(* IEC 61131-3 sources: Elmo_Master/Lasal_PRG/Elmo_EtherCAT_Test_4Axis/Class/LMCDiagnosticsService (part 3) *)

			32:
				mailboxResult := InputLatch.SubmitDs402HomeControl(
					OperationToken:=Ds402HomeState[101]$UDINT,
					AxisReference:=axisReference, Command:=4);
				if mailboxResult = 0 then
					Ds402HomeState[117] := 0;
					Ds402HomeState[112] := currentCycle$DINT;
					Ds402HomeState[92] := 34;
				elsif mailboxResult = 1 then
					Ds402HomeState[92] := 33;
				else
					failure := TRUE;
					failureDetail := 11;
					failureNative := TO_UDINT(0 - mailboxResult);
				end_if;

			33:
				mailboxResult := InputLatch.GetDs402HomeControlState(
					OperationToken:=Ds402HomeState[101]$UDINT);
				if mailboxResult = 0 then
					Ds402HomeState[117] := 0;
					Ds402HomeState[112] := currentCycle$DINT;
					Ds402HomeState[92] := 34;
				elsif mailboxResult <> 1 then
					failure := TRUE;
					failureDetail := 11;
					failureNative := TO_UDINT(0 - mailboxResult);
				end_if;

			34:
				if newCycle &
					(currentCycle <> Ds402HomeState[112]$UDINT) then
					if (Ds402HomeState[94] <> 0) |
						(Ds402HomeState[113] <> 0) |
						(Ds402HomeState[116] <> 0) |
						(Ds402HomeState[117] <> 0) |
						(Ds402HomeState[127] <> 0) |
						((statusWord and 0x0008) <> 0) |
						((statusWord and 0x2000) <> 0) |
						((baseState <> 0x0040) & (baseState <> 0x0021) &
						 (baseState <> 0x0023) & (baseState <> 0x0027)) |
						(actualPosition <> 0) then
						failure := TRUE;
						failureNative := 24;
					else
						Ds402HomeState[106] := 2;
						Ds402HomeState[107] := 0;
						Ds402HomeState[108] := 0;
						Ds402HomeState[recordBase + 14] := 0;
						Ds402HomeState[recordBase + 15] := 0;
						Ds402HomeState[recordBase + 16] := 0;
						Ds402HomeState[recordBase + 20] := currentCycle$DINT;
						Ds402HomeState[recordBase + 21] := 0;
						ownerResult := -1;
						if IsClientConnected(#AxisOwnership) then
							ownerResult :=
								AxisOwnership.PublishAxisOwnershipDs402Receipt(
								AxisMask:=axisMask,
								AdmissionToken:=admissionToken,
								OwnerGeneration:=ownerGeneration,
								ReportKind:=
									LMC_DIAG_OWNER_REPORT_TERMINAL_SUCCESS,
								ReportValue0:=0,
								ReportValue1:=0,
								ObservationCycle:=currentCycle,
								pDs402State:=#Ds402HomeState[0],
								Ds402StateSize:=sizeof(Ds402HomeState));
						end_if;
						if ownerResult = 0 then
							Ds402HomeState[125] := 2;
							ownerResult :=
								AxisOwnership.PublishAxisOwnershipDs402Receipt(
									AxisMask:=axisMask,
									AdmissionToken:=admissionToken,
									OwnerGeneration:=ownerGeneration,
									ReportKind:=
										LMC_DIAG_OWNER_REPORT_TERMINAL_SUCCESS,
									ReportValue0:=0,
									ReportValue1:=0,
									ObservationCycle:=currentCycle,
									pDs402State:=#Ds402HomeState[0],
									Ds402StateSize:=sizeof(Ds402HomeState));
							if ownerResult = 1 then
								Ds402HomeState[92] :=
									LMC_DIAG_DS402_STAGE_FINALIZE;
							elsif ownerResult <> 0 then
								Ds402HomeState[92] := 101;
							end_if;
							RETURN;
						elsif ownerResult = 1 then
							Ds402HomeState[92] := LMC_DIAG_DS402_STAGE_FINALIZE;
							RETURN;
						else
							Ds402HomeState[92] := 101;
						end_if;
					end_if;
				end_if;
		end_case;
	end_if;

	// SDO start stages use one persistent executor at a time.
	stage := Ds402HomeState[92];
	startSdo := FALSE;
	sdoIsWrite := FALSE;
	sdoIndex := 0;
	homeSdoSubIndex := 0;
	sdoLength := 0;
	sdoData := 0;
	nextStage := stage;
	if (failure = FALSE) & (stage < 90) then
		case stage of
			2:
				startSdo := TRUE; sdoIndex := 0x6061;
				sdoLength := 1; nextStage := 3;
			4:
				startSdo := TRUE; sdoIsWrite := TRUE; sdoIndex := 0x607C;
				sdoLength := 4; sdoData := Ds402HomeState[recordBase + 10]$UDINT;
				nextStage := 5;
			6:
				startSdo := TRUE; sdoIsWrite := TRUE; sdoIndex := 0x6098;
				sdoLength := 1; sdoData := Ds402HomeState[recordBase + 9]$UDINT;
				nextStage := 7;
			16:
				startSdo := TRUE; sdoIsWrite := TRUE; sdoIndex := 0x6060;
				sdoLength := 1; sdoData := 6; nextStage := 17;
			18:
				startSdo := TRUE; sdoIndex := 0x6061;
				sdoLength := 1; nextStage := 19;
			28:
				startSdo := TRUE; sdoIsWrite := TRUE; sdoIndex := 0x6060;
				sdoLength := 1; sdoData := 8; nextStage := 29;
			30:
				startSdo := TRUE; sdoIndex := 0x6061;
				sdoLength := 1; nextStage := 31;
		end_case;
	end_if;

	if startSdo then
		if IsClientConnected(#AxisOwnership) = FALSE then
			failure := TRUE;
			failureNative := 24;
		else
			ownerResult := AxisOwnership.ValidateAxisOwnership(
				CommandId:=0x7D15,
				Reference:=axisReference,
				ExpectedAxisMask:=axisMask,
				OwnerKind:=LMC_DIAG_OWNER_KIND_DS402_HOME,
				ResourceKind:=LMC_DIAG_RESOURCE_DS402_HOME,
				AdmissionMode:=LMC_DIAG_ADMISSION_LIFECYCLE,
				CallerSessionEpoch:=ds402ProcessOwnerSessionEpoch,
				RequestSequence:=ownerRequestSequence,
				AdmissionToken:=admissionToken,
				OwnerGeneration:=ownerGeneration,
				RequiredPhase:=LMC_DIAG_OWNER_PHASE_ACTIVE);
			if ownerResult <> 0 then
				failure := TRUE;
				failureNative := TO_UDINT(0 - ownerResult);
			elsif Ds402HomeState[126] = 0 then
					ownerResult := AxisOwnership.PublishAxisOwnership(
						AxisMask:=axisMask,
						AdmissionToken:=admissionToken,
						OwnerGeneration:=ownerGeneration,
						ReportKind:=LMC_DIAG_OWNER_REPORT_DISPATCH,
						ReportValue0:=TO_UDINT(sdoIndex),
						ReportValue1:=Ds402HomeState[101]$UDINT,
						ObservationCycle:=currentCycle);
				if ownerResult = 0 then
					Ds402HomeState[126] := 1;
				else
					failure := TRUE;
					failureNative := TO_UDINT(0 - ownerResult);
				end_if;
			end_if;
		end_if;
	end_if;

	if startSdo & (failure = FALSE) then
		executorConnected := FALSE;
		executorReusable := FALSE;
		case axisReference of
			1:
				executorConnected := IsClientConnected(#SdoAxis1) <> 0;
				if executorConnected then
					executorReusable := SdoAxis1.IsReusable();
				end_if;
			2:
				executorConnected := IsClientConnected(#SdoAxis2) <> 0;
				if executorConnected then
					executorReusable := SdoAxis2.IsReusable();
				end_if;
			3:
				executorConnected := IsClientConnected(#SdoAxis3) <> 0;
				if executorConnected then
					executorReusable := SdoAxis3.IsReusable();
				end_if;
			4:
				executorConnected := IsClientConnected(#SdoAxis4) <> 0;
				if executorConnected then
					executorReusable := SdoAxis4.IsReusable();
				end_if;
		end_case;
		if (executorConnected = FALSE) | (executorReusable = FALSE) then
			failure := TRUE;
			failureNative := 24;
		else
			sdoToken := Ds402HomeState[99]$UDINT + 1;
			if sdoToken = 0 then
				sdoToken := 1;
			end_if;
			Ds402HomeState[99] := sdoToken$DINT;
			Ds402HomeState[95] := 0;
			if sdoIsWrite then
				Ds402HomeState[95] := 1;
			end_if;
			Ds402HomeState[96] := sdoIndex$DINT;
			Ds402HomeState[97] := homeSdoSubIndex$DINT;
			Ds402HomeState[98] := sdoLength$DINT;
			Ds402HomeState[100] := sdoData$DINT;
			startCycle := Ds402HomeState[recordBase + 19]$UDINT;
			timeoutMs := Ds402HomeState[recordBase + 13]$UDINT;
			elapsedCycles := serviceNow - serviceStart;
			remainingMs := 1;
			if elapsedCycles < timeoutMs then
				remainingMs := timeoutMs - elapsedCycles;
			end_if;
			if remainingMs > 60000 then
				remainingMs := 60000;
			end_if;
			startResult := ERROR;
			case axisReference of
				1:
					if sdoIsWrite then
						startResult := SdoAxis1.TryStartWrite(sdoToken, sdoIndex,
							homeSdoSubIndex, (#sdoData)$^USINT, sdoLength, remainingMs);
					else
						startResult := SdoAxis1.TryStartRead(sdoToken, sdoIndex,
							homeSdoSubIndex, sdoLength, remainingMs);
					end_if;
				2:
					if sdoIsWrite then
						startResult := SdoAxis2.TryStartWrite(sdoToken, sdoIndex,
							homeSdoSubIndex, (#sdoData)$^USINT, sdoLength, remainingMs);
					else
						startResult := SdoAxis2.TryStartRead(sdoToken, sdoIndex,
							homeSdoSubIndex, sdoLength, remainingMs);
					end_if;
				3:
					if sdoIsWrite then
						startResult := SdoAxis3.TryStartWrite(sdoToken, sdoIndex,
							homeSdoSubIndex, (#sdoData)$^USINT, sdoLength, remainingMs);
					else
						startResult := SdoAxis3.TryStartRead(sdoToken, sdoIndex,
							homeSdoSubIndex, sdoLength, remainingMs);
					end_if;
				4:
					if sdoIsWrite then
						startResult := SdoAxis4.TryStartWrite(sdoToken, sdoIndex,
							homeSdoSubIndex, (#sdoData)$^USINT, sdoLength, remainingMs);
					else
						startResult := SdoAxis4.TryStartRead(sdoToken, sdoIndex,
							homeSdoSubIndex, sdoLength, remainingMs);
					end_if;
			end_case;
			if startResult = READY then
				// Once the mode-6 write is accepted, cleanup must assume it may
				// have reached the drive even if its callback is later lost.
				if stage = 16 then
					Ds402HomeState[116] := 1;
				end_if;
				Ds402HomeState[94] := 1;
				Ds402HomeState[92] := nextStage;
			else
				failure := TRUE;
				failureNative := 24;
			end_if;
		end_if;
	end_if;

	stage := Ds402HomeState[92];
	waitSdo := (stage = 3) | (stage = 5) | (stage = 7) |
		(stage = 17) | (stage = 19) | (stage = 29) | (stage = 31);
	if (failure = FALSE) & waitSdo then
		completionResult := -2;
		case axisReference of
			1:
				if IsClientConnected(#SdoAxis1) then
					completionResult := SdoAxis1.CopyCompletion(
						Ds402HomeState[99]$UDINT, #completion, sizeof(completion));
				end_if;
			2:
				if IsClientConnected(#SdoAxis2) then
					completionResult := SdoAxis2.CopyCompletion(
						Ds402HomeState[99]$UDINT, #completion, sizeof(completion));
				end_if;
			3:
				if IsClientConnected(#SdoAxis3) then
					completionResult := SdoAxis3.CopyCompletion(
						Ds402HomeState[99]$UDINT, #completion, sizeof(completion));
				end_if;
			4:
				if IsClientConnected(#SdoAxis4) then
					completionResult := SdoAxis4.CopyCompletion(
						Ds402HomeState[99]$UDINT, #completion, sizeof(completion));
				end_if;
		end_case;
		if completionResult = 0 then
			Ds402HomeState[94] := 0;
			if (completion.ValidationCode <> 0) | (completion.OsResult <> 0) |
				(completion.AbortCode <> 0) |
				(completion.ObjectIndex <> Ds402HomeState[96]$UINT) |
				(completion.SubIndex <> Ds402HomeState[97]$USINT) |
				(completion.ActualLength <> Ds402HomeState[98]$UDINT) |
				(completion.IsWrite <> Ds402HomeState[95]$USINT) then
				failure := TRUE;
				if completion.AbortCode <> 0 then
					failureNative := completion.AbortCode;
				elsif completion.OsResult <> 0 then
					failureNative := completion.OsResult$UDINT;
				else
					failureNative := completion.ValidationCode;
				end_if;
			else
				case stage of
					3:
						if (completion.Data and 0xFF) <> 8 then
							failure := TRUE; failureNative := completion.Data;
						else
							Ds402HomeState[105] := 8; Ds402HomeState[92] := 4;
						end_if;
					5: Ds402HomeState[92] := 6;
					7: Ds402HomeState[92] := 14;
					17:
						Ds402HomeState[116] := 1; Ds402HomeState[92] := 18;
					19:
						if (completion.Data and 0xFF) <> 6 then
							failure := TRUE; failureNative := completion.Data;
						else
							Ds402HomeState[92] := 20;
						end_if;
					29: Ds402HomeState[92] := 30;
					31:
						if (completion.Data and 0xFF) <> 8 then
							failure := TRUE; failureNative := completion.Data;
						else
							Ds402HomeState[116] := 0; Ds402HomeState[92] := 32;
						end_if;
				end_case;
			end_if;
		elsif (completionResult <> -2) & (completionResult <> -3) then
			failure := TRUE;
			failureNative := TO_UDINT(0 - completionResult);
		end_if;
	end_if;

	if failure then
		if Ds402HomeState[94] <> 0 then
			orphanResult := -1;
			case axisReference of
				1:
					if IsClientConnected(#SdoAxis1) then
						orphanResult := SdoAxis1.MarkOrphan(Ds402HomeState[99]$UDINT);
					end_if;
				2:
					if IsClientConnected(#SdoAxis2) then
						orphanResult := SdoAxis2.MarkOrphan(Ds402HomeState[99]$UDINT);
					end_if;
				3:
					if IsClientConnected(#SdoAxis3) then
						orphanResult := SdoAxis3.MarkOrphan(Ds402HomeState[99]$UDINT);
					end_if;
				4:
					if IsClientConnected(#SdoAxis4) then
						orphanResult := SdoAxis4.MarkOrphan(Ds402HomeState[99]$UDINT);
					end_if;
			end_case;
			// -2 can mean that the exact result won the timeout race. Keep the
			// executor in the cleanup drain path so a ready result is consumed.
			if (orphanResult = 0) | (orphanResult = -2) then
				Ds402HomeState[94] := 0;
				Ds402HomeState[113] := 1;
				Ds402HomeState[127] := 0;
			else
				// Keep the pending token and remember that exact retirement failed.
				Ds402HomeState[127] := 1;
			end_if;
		end_if;
		if preemptionCleanup then
			Ds402HomeState[106] := 4;
		else
			Ds402HomeState[106] := 3;
		end_if;
		Ds402HomeState[107] := failureDetail$DINT;
		Ds402HomeState[108] := failureNative$DINT;
		Ds402HomeState[112] := currentCycle$DINT;
		Ds402HomeState[119]$UDINT := serviceNow;
		Ds402HomeState[92] := 90;
		RETURN;
	end_if;

	// Failure cleanup attempts bit 4 low, setpoint alignment, CSP restore and RT
	// release. Timeout never claims that any of those cleanup steps completed.
	stage := Ds402HomeState[92];
	if stage < 90 then
		RETURN;
	end_if;
	if preemptionCleanup then
		HandleAxisDs402HomeCleanupStages(
			Stage:=stage,
			AxisReference:=axisReference,
			AxisMask:=axisMask,
			AdmissionToken:=admissionToken,
			OwnerGeneration:=ownerGeneration,
			Ds402ProcessOwnerSessionEpoch:=ds402ProcessOwnerSessionEpoch,
			OwnerRequestSequence:=ownerRequestSequence,
			SafetyAdmissionToken:=safetyAdmissionToken,
			SafetyOwnerGeneration:=safetyOwnerGeneration,
			InitialCurrentCycle:=currentCycle,
			ServiceNow:=serviceNow,
			ActualPosition:=actualPosition,
			PreemptionCleanup:=TRUE);
	else
		HandleAxisDs402HomeCleanupStages(
			Stage:=stage,
			AxisReference:=axisReference,
			AxisMask:=axisMask,
			AdmissionToken:=admissionToken,
			OwnerGeneration:=ownerGeneration,
			Ds402ProcessOwnerSessionEpoch:=ds402ProcessOwnerSessionEpoch,
			OwnerRequestSequence:=ownerRequestSequence,
			SafetyAdmissionToken:=0,
			SafetyOwnerGeneration:=0,
			InitialCurrentCycle:=currentCycle,
			ServiceNow:=serviceNow,
			ActualPosition:=actualPosition,
			PreemptionCleanup:=FALSE);
	end_if;

END_FUNCTION

FUNCTION LMCDiagnosticsService::HandleAxisDs402HomeReceiptStages
	VAR_INPUT
		Stage 	: DINT;
	END_VAR
	VAR_OUTPUT
		Result 	: DINT;
	END_VAR
	VAR
		activeIndex, recordBase : DINT;
		axisReference : UINT;
		axisMask, admissionToken, ownerGeneration : UDINT;
		ds402ProcessOwnerSessionEpoch, ownerRequestSequence : UDINT;
		receiptGeneration : UDINT;
		ownerResult, receiptResult, receiptKind, receiptPhase : DINT;
		terminalRecordState : DINT;
	END_VAR

	Result := 1;
	if stage = LMC_DIAG_DS402_STAGE_INTENT_DISCARD_CLEAR then
		activeIndex := Ds402HomeState[93];
		if (activeIndex < 0) | (activeIndex > 3) |
			(sizeof(Ds402HomeState) <> 512) then
			Ds402HomeState[92] := 101;
			RETURN;
		end_if;
		recordBase := activeIndex * 23;
		// Stage 86 keeps the axis selector authoritative until this idempotent
		// record clear is complete. Runtime WAL bytes remain invalid under stage 0
		// and are replaced by the next preflight.
		_memset(dest:=#Ds402HomeState[recordBase], usByte:=0, cntr:=92);
		Ds402HomeState[92] := 0;
		RETURN;
	end_if;
	if stage = LMC_DIAG_DS402_STAGE_RESERVE_INTENT then
		activeIndex := Ds402HomeState[93];
		if (activeIndex < 0) | (activeIndex > 3) |
			(sizeof(Ds402HomeState) <> 512) then
			Ds402HomeState[92] := 101;
			RETURN;
		end_if;
		recordBase := activeIndex * 23;
		axisMask := TO_UDINT(1) shl TO_UDINT(activeIndex);
		if IsClientConnected(#AxisOwnership) = FALSE then
			RETURN;
		end_if;
		// Tokenless mode is confined to stage 87 rollback resolution. The
		// provider either adopts one exact RESERVED tuple, proves absence/later
		// ownership, or leaves the intent fail-closed.
		receiptResult := AxisOwnership.PublishAxisOwnershipDs402Receipt(
			AxisMask:=axisMask,
			AdmissionToken:=0,
			OwnerGeneration:=0,
			ReportKind:=LMC_DIAG_DS402_RECEIPT_ROLLBACK,
			ReportValue0:=0,
			ReportValue1:=0,
			ObservationCycle:=Ds402HomeState[118]$UDINT,
			pDs402State:=#Ds402HomeState[0],
			Ds402StateSize:=sizeof(Ds402HomeState));
		if receiptResult = 1 then
			// Commit record cleanup before touching any selector or WAL byte.
			Ds402HomeState[92] :=
				LMC_DIAG_DS402_STAGE_INTENT_DISCARD_CLEAR;
		elsif receiptResult = 2 then
			// Preserve only an untouched raw tombstone. Once adoption or the record
			// bridge was published, commit a durable record-clear cleanup first.
			if (Ds402HomeState[119]$UDINT =
				LMC_DIAG_DS402_INTENT_ADOPT_MAGIC) |
				(Ds402HomeState[recordBase] = 1) then
				Ds402HomeState[92] :=
					LMC_DIAG_DS402_STAGE_INTENT_DISCARD_CLEAR;
			elsif Ds402HomeState[recordBase]$UDINT <>
				Ds402HomeState[115]$UDINT then
				Ds402HomeState[92] := 101;
				RETURN;
			else
				// No local record changed. Stage 0 invalidates the retained WAL in one
				// commit; the next preflight overwrites it before reuse.
				Ds402HomeState[92] := 0;
			end_if;
		elsif receiptResult = -1 then
			// A transient result retains the durable intent indefinitely.
		elsif receiptResult <> 0 then
			Ds402HomeState[92] := 101;
		end_if;
		RETURN;
	end_if;
	if stage = 0 then
		RETURN;
	end_if;
	activeIndex := Ds402HomeState[93];
	admissionToken := Ds402HomeState[122]$UDINT;
	ownerGeneration := Ds402HomeState[123]$UDINT;
	if (activeIndex < 0) | (activeIndex > 3) |
		(sizeof(Ds402HomeState) <> 512) then
		Ds402HomeState[92] := 101;
		RETURN;
	end_if;
	recordBase := activeIndex * 23;
	axisMask := TO_UDINT(1) shl TO_UDINT(activeIndex);
	receiptPhase := Ds402HomeState[125];
	receiptGeneration := Ds402HomeState[127]$UDINT;

	if stage = LMC_DIAG_DS402_STAGE_FINALIZE then
		receiptKind := Ds402HomeState[126];
		if (Ds402HomeState[124]$UDINT <> LMC_DIAG_DS402_RECEIPT_MAGIC) |
			(receiptPhase <> LMC_DIAG_DS402_RECEIPT_COMPLETE) |
			(receiptGeneration = 0) |
			(receiptGeneration <> Ds402HomeState[109]$UDINT) |
			(admissionToken = 0) | (ownerGeneration = 0) then
			Ds402HomeState[92] := 101;
			RETURN;
		end_if;
		case receiptKind of
			LMC_DIAG_DS402_RECEIPT_ROLLBACK:
				if (Ds402HomeState[106] <> 0) |
					((Ds402HomeState[recordBase] <> 0) &
					 (Ds402HomeState[recordBase] <> 1)) |
					((Ds402HomeState[recordBase + 22]$UDINT <> 0) &
					 (Ds402HomeState[recordBase + 22]$UDINT <>
					  receiptGeneration)) then
					Ds402HomeState[92] := 101;
					RETURN;
				end_if;
				_memset(dest:=#Ds402HomeState[recordBase],
					usByte:=0, cntr:=92);
			LMC_DIAG_OWNER_REPORT_TERMINAL_SUCCESS,
			LMC_DIAG_OWNER_REPORT_TERMINAL_SAFE_FAILURE:
				terminalRecordState := Ds402HomeState[106];
				if (((receiptKind = LMC_DIAG_OWNER_REPORT_TERMINAL_SUCCESS) &
					  (terminalRecordState <> 2)) |
					 ((receiptKind =
					   LMC_DIAG_OWNER_REPORT_TERMINAL_SAFE_FAILURE) &
					  (terminalRecordState <> 3))) |
					(Ds402HomeState[recordBase + 22]$UDINT <>
					 receiptGeneration) |
					((Ds402HomeState[recordBase] <> 1) &
					 (Ds402HomeState[recordBase] <> terminalRecordState)) then
					Ds402HomeState[92] := 101;
					RETURN;
				end_if;
				Ds402HomeState[101] := 0;
				Ds402HomeState[recordBase] := terminalRecordState;
		else
			Ds402HomeState[92] := 101;
			RETURN;
		end_case;
		// The local lifecycle stage is the final publication word.
		Ds402HomeState[92] := 0;
		RETURN;
	end_if;

	if Ds402HomeState[124]$UDINT = LMC_DIAG_DS402_RECEIPT_MAGIC then
		if receiptGeneration = 0 then
			case stage of
				LMC_DIAG_DS402_STAGE_ROLLBACK_PREPARED:
					receiptKind := LMC_DIAG_DS402_RECEIPT_ROLLBACK;
				89: receiptKind := LMC_DIAG_DS402_RECEIPT_ROLLBACK;
				34: receiptKind := LMC_DIAG_OWNER_REPORT_TERMINAL_SUCCESS;
				100: receiptKind :=
					LMC_DIAG_OWNER_REPORT_TERMINAL_SAFE_FAILURE;
			else
				Ds402HomeState[92] := 101;
				RETURN;
			end_case;
		else
			receiptKind := Ds402HomeState[126];
		end_if;
		receiptResult := -1;
		if IsClientConnected(#AxisOwnership) = FALSE then
			RETURN;
		end_if;
		receiptResult := AxisOwnership.PublishAxisOwnershipDs402Receipt(
			AxisMask:=axisMask,
			AdmissionToken:=admissionToken,
			OwnerGeneration:=ownerGeneration,
			ReportKind:=TO_UINT(receiptKind),
			ReportValue0:=Ds402HomeState[107]$UDINT,
			ReportValue1:=Ds402HomeState[108]$UDINT,
			ObservationCycle:=Ds402HomeState[110]$UDINT,
			pDs402State:=#Ds402HomeState[0],
			Ds402StateSize:=sizeof(Ds402HomeState));
		if receiptResult = 0 then
			if Ds402HomeState[125] = LMC_DIAG_DS402_RECEIPT_PREPARED then
				Ds402HomeState[125] := 2;
			end_if;
			if IsClientConnected(#AxisOwnership) = FALSE then
				RETURN;
			end_if;
			receiptResult :=
				AxisOwnership.PublishAxisOwnershipDs402Receipt(
					AxisMask:=axisMask,
					AdmissionToken:=admissionToken,
					OwnerGeneration:=ownerGeneration,
					ReportKind:=TO_UINT(receiptKind),
					ReportValue0:=Ds402HomeState[107]$UDINT,
					ReportValue1:=Ds402HomeState[108]$UDINT,
					ObservationCycle:=Ds402HomeState[110]$UDINT,
					pDs402State:=#Ds402HomeState[0],
					Ds402StateSize:=sizeof(Ds402HomeState));
			if receiptResult = 1 then
				Ds402HomeState[92] := LMC_DIAG_DS402_STAGE_FINALIZE;
			elsif (receiptResult <> 0) & (receiptResult <> -1) then
				Ds402HomeState[92] := 101;
			end_if;
		elsif receiptResult = 1 then
			Ds402HomeState[92] := LMC_DIAG_DS402_STAGE_FINALIZE;
		elsif receiptResult <> -1 then
			Ds402HomeState[92] := 101;
		end_if;
		RETURN;
	end_if;

	if stage = LMC_DIAG_DS402_STAGE_ROLLBACK_PREPARED then
		// This state is rollback-only. It must never warm-resume into Commit.
		receiptResult := -1;
		if IsClientConnected(#AxisOwnership) = FALSE then
			RETURN;
		end_if;
		receiptResult := AxisOwnership.PublishAxisOwnershipDs402Receipt(
			AxisMask:=axisMask,
			AdmissionToken:=admissionToken,
			OwnerGeneration:=ownerGeneration,
			ReportKind:=LMC_DIAG_DS402_RECEIPT_ROLLBACK,
			ReportValue0:=0,
			ReportValue1:=0,
			ObservationCycle:=Ds402HomeState[110]$UDINT,
			pDs402State:=#Ds402HomeState[0],
			Ds402StateSize:=sizeof(Ds402HomeState));
		if receiptResult = 0 then
			if Ds402HomeState[125] =
				LMC_DIAG_DS402_RECEIPT_PREPARED then
				Ds402HomeState[125] := 2;
			end_if;
			if IsClientConnected(#AxisOwnership) = FALSE then
				RETURN;
			end_if;
			receiptResult :=
				AxisOwnership.PublishAxisOwnershipDs402Receipt(
					AxisMask:=axisMask,
					AdmissionToken:=admissionToken,
					OwnerGeneration:=ownerGeneration,
					ReportKind:=LMC_DIAG_DS402_RECEIPT_ROLLBACK,
					ReportValue0:=0,
					ReportValue1:=0,
					ObservationCycle:=Ds402HomeState[110]$UDINT,
					pDs402State:=#Ds402HomeState[0],
					Ds402StateSize:=sizeof(Ds402HomeState));
			if receiptResult = 1 then
				Ds402HomeState[92] := LMC_DIAG_DS402_STAGE_FINALIZE;
			elsif (receiptResult <> 0) & (receiptResult <> -1) then
				Ds402HomeState[92] := 101;
			end_if;
		elsif receiptResult = 1 then
			Ds402HomeState[92] := LMC_DIAG_DS402_STAGE_FINALIZE;
		elsif receiptResult <> -1 then
			Ds402HomeState[92] := 101;
		end_if;
		RETURN;
	end_if;

	if stage = 101 then
		// Quarantine is terminal for this cyclic processor.
		RETURN;
	end_if;
	if stage = 89 then
		if (activeIndex < 0) | (activeIndex > 3) |
			(sizeof(Ds402HomeState) <> 512) then
			Ds402HomeState[92] := 101;
			RETURN;
		end_if;
		axisReference := TO_UINT(activeIndex + 1);
		recordBase := activeIndex * 23;
		axisMask := Ds402HomeState[124]$UDINT;
		ds402ProcessOwnerSessionEpoch := Ds402HomeState[120]$UDINT;
		ownerRequestSequence := Ds402HomeState[121]$UDINT;
		if (axisMask <> (TO_UDINT(1) shl TO_UDINT(activeIndex))) |
			(ds402ProcessOwnerSessionEpoch = 0) |
			(ownerRequestSequence = 0) | (admissionToken = 0) |
			(ownerGeneration = 0) |
			(Ds402HomeState[recordBase] <> 1) |
			(Ds402HomeState[recordBase + 1] <> 1) |
			(Ds402HomeState[recordBase + 2]$UDINT <>
			 GetDiagnosticsBootId()) |
			(Ds402HomeState[recordBase + 3]$UDINT <>
			 LMC_DIAG_MAP_REVISION) |
			(Ds402HomeState[recordBase + 4] = 0) |
			((Ds402HomeState[recordBase + 5] = 0) &
			 (Ds402HomeState[recordBase + 6] = 0) &
			 (Ds402HomeState[recordBase + 7] = 0) &
			 (Ds402HomeState[recordBase + 8] = 0)) |
			(Ds402HomeState[recordBase + 9] <> 37) |
			(Ds402HomeState[recordBase + 10] <> 0) |
			(Ds402HomeState[recordBase + 11] <> 0) |
			(Ds402HomeState[recordBase + 12] <> 0) |
			(Ds402HomeState[recordBase + 13] = 0) |
			(Ds402HomeState[recordBase + 14] <> 0) |
			(Ds402HomeState[recordBase + 15] <> 0) |
			(Ds402HomeState[recordBase + 16] <> 0) |
			(Ds402HomeState[recordBase + 19] = 0) |
			(Ds402HomeState[recordBase + 20] <> 0) |
			(Ds402HomeState[recordBase + 21] <> 0) |
			(Ds402HomeState[recordBase + 22] = 0) |
			(Ds402HomeState[94] <> 0) |
			(Ds402HomeState[95] <> 0) |
			(Ds402HomeState[96] <> 0) |
			(Ds402HomeState[97] <> 0) |
			(Ds402HomeState[98] <> 0) |
			(Ds402HomeState[100] <> 0) |
			(Ds402HomeState[109] <>
			 Ds402HomeState[recordBase + 22]) |
			(Ds402HomeState[99] <>
			 Ds402HomeState[recordBase + 22]) |
			(Ds402HomeState[101] <>
			 Ds402HomeState[recordBase + 22]) |
			(Ds402HomeState[102] <>
			 Ds402HomeState[recordBase + 18]) |
			(Ds402HomeState[103] <> 1) |
			(Ds402HomeState[104] <> 0) |
			(Ds402HomeState[105] <> 8) |
			(Ds402HomeState[106] <> 0) |
			(Ds402HomeState[107] <> 0) |
			(Ds402HomeState[108] <> 0) |
			(Ds402HomeState[110] <>
			 Ds402HomeState[recordBase + 19]) |
			(Ds402HomeState[111] <> 0) |
			(Ds402HomeState[112] <> 0) |
			(Ds402HomeState[113] <> 0) |
			(Ds402HomeState[114] <>
			 Ds402HomeState[recordBase + 17]) |
			(Ds402HomeState[115] <>
			 Ds402HomeState[recordBase + 18]) |
			(Ds402HomeState[116] <> 0) |
			(Ds402HomeState[117] <> 0) |
			(Ds402HomeState[119] <> 0) |
			(Ds402HomeState[126] <> 0) |
			(Ds402HomeState[127] <> 0) |
			((Ds402HomeState[125] <> 1) &
			 (Ds402HomeState[125] <> 2)) then
			Ds402HomeState[92] := 101;
			RETURN;
		end_if;
		if IsClientConnected(#AxisOwnership) = FALSE then
			RETURN;
		end_if;

		// Commit may already have completed before the local phase was advanced.
		ownerResult := AxisOwnership.ValidateAxisOwnership(
			CommandId:=0x7D15,
			Reference:=axisReference,
			ExpectedAxisMask:=axisMask,
			OwnerKind:=LMC_DIAG_OWNER_KIND_DS402_HOME,
			ResourceKind:=LMC_DIAG_RESOURCE_DS402_HOME,
			AdmissionMode:=LMC_DIAG_ADMISSION_LIFECYCLE,
			CallerSessionEpoch:=ds402ProcessOwnerSessionEpoch,
			RequestSequence:=ownerRequestSequence,
			AdmissionToken:=admissionToken,
			OwnerGeneration:=ownerGeneration,
			RequiredPhase:=LMC_DIAG_OWNER_PHASE_ACTIVE);
		if ownerResult = 0 then
			Ds402HomeState[125] := 2;
			Ds402HomeState[92] := 1;
			RETURN;
		end_if;

		ownerResult := AxisOwnership.ValidateAxisOwnership(
			CommandId:=0x7D15,
			Reference:=axisReference,
			ExpectedAxisMask:=axisMask,
			OwnerKind:=LMC_DIAG_OWNER_KIND_DS402_HOME,
			ResourceKind:=LMC_DIAG_RESOURCE_DS402_HOME,
			AdmissionMode:=LMC_DIAG_ADMISSION_LIFECYCLE,
			CallerSessionEpoch:=ds402ProcessOwnerSessionEpoch,
			RequestSequence:=ownerRequestSequence,
			AdmissionToken:=admissionToken,
			OwnerGeneration:=ownerGeneration,
			RequiredPhase:=LMC_DIAG_OWNER_PHASE_RESERVED);
		if (ownerResult = 0) & (Ds402HomeState[125] = 1) then
			ownerResult := AxisOwnership.CommitAxisOwnership(
				CommandId:=0x7D15,
				Reference:=axisReference,
				ExpectedAxisMask:=axisMask,
				CallerSessionEpoch:=ds402ProcessOwnerSessionEpoch,
				RequestSequence:=ownerRequestSequence,
				AdmissionToken:=admissionToken,
				OwnerGeneration:=ownerGeneration);
			if ownerResult = 0 then
				Ds402HomeState[125] := 2;
				Ds402HomeState[92] := 1;
				RETURN;
			end_if;
			ownerResult := AxisOwnership.ValidateAxisOwnership(
				CommandId:=0x7D15,
				Reference:=axisReference,
				ExpectedAxisMask:=axisMask,
				OwnerKind:=LMC_DIAG_OWNER_KIND_DS402_HOME,
				ResourceKind:=LMC_DIAG_RESOURCE_DS402_HOME,
				AdmissionMode:=LMC_DIAG_ADMISSION_LIFECYCLE,
				CallerSessionEpoch:=ds402ProcessOwnerSessionEpoch,
				RequestSequence:=ownerRequestSequence,
				AdmissionToken:=admissionToken,
				OwnerGeneration:=ownerGeneration,
				RequiredPhase:=LMC_DIAG_OWNER_PHASE_ACTIVE);
			if ownerResult = 0 then
				Ds402HomeState[125] := 2;
				Ds402HomeState[92] := 1;
				RETURN;
			end_if;
		end_if;

		receiptResult := AxisOwnership.PublishAxisOwnershipDs402Receipt(
			AxisMask:=axisMask,
			AdmissionToken:=admissionToken,
			OwnerGeneration:=ownerGeneration,
			ReportKind:=LMC_DIAG_DS402_RECEIPT_ROLLBACK,
			ReportValue0:=0,
			ReportValue1:=0,
			ObservationCycle:=Ds402HomeState[110]$UDINT,
			pDs402State:=#Ds402HomeState[0],
			Ds402StateSize:=sizeof(Ds402HomeState));
		if receiptResult = 0 then
			if Ds402HomeState[125] =
				LMC_DIAG_DS402_RECEIPT_PREPARED then
				Ds402HomeState[125] := 2;
			end_if;
			receiptResult := AxisOwnership.PublishAxisOwnershipDs402Receipt(
				AxisMask:=axisMask,
				AdmissionToken:=admissionToken,
				OwnerGeneration:=ownerGeneration,
				ReportKind:=LMC_DIAG_DS402_RECEIPT_ROLLBACK,
				ReportValue0:=0,
				ReportValue1:=0,
				ObservationCycle:=Ds402HomeState[110]$UDINT,
				pDs402State:=#Ds402HomeState[0],
				Ds402StateSize:=sizeof(Ds402HomeState));
			if receiptResult = 1 then
				Ds402HomeState[92] := LMC_DIAG_DS402_STAGE_FINALIZE;
			elsif (receiptResult <> 0) & (receiptResult <> -1) then
				Ds402HomeState[92] := 101;
			end_if;
		elsif receiptResult = 1 then
			Ds402HomeState[92] := LMC_DIAG_DS402_STAGE_FINALIZE;
		elsif receiptResult <> -1 then
			Ds402HomeState[92] := 101;
		end_if;
		RETURN;
	end_if;
	Result := 0;

END_FUNCTION

FUNCTION LMCDiagnosticsService::HandleAxisDs402HomeCleanupStages
	VAR_INPUT
		Stage 	: DINT;
		AxisReference 	: UINT;
		AxisMask 	: UDINT;
		AdmissionToken 	: UDINT;
		OwnerGeneration 	: UDINT;
		Ds402ProcessOwnerSessionEpoch 	: UDINT;
		OwnerRequestSequence 	: UDINT;
		SafetyAdmissionToken 	: UDINT;
		SafetyOwnerGeneration 	: UDINT;
		InitialCurrentCycle 	: UDINT;
		ServiceNow 	: UDINT;
		ActualPosition 	: DINT;
		PreemptionCleanup 	: BOOL;
	END_VAR
	VAR
		completion : LMCSdoExecutor::LMCSdoExecutorResult;
		recordBase : DINT;
		preemptionCleanupKind : UINT;
		currentCycle, cleanupStart, sdoToken, sdoData : UDINT;
		completionResult, mailboxResult, orphanResult, ownerResult : DINT;
		startResult : iprStates;
		executorConnected, executorReusable, cleanupExpired : BOOL;
	END_VAR

	currentCycle := InitialCurrentCycle;
	recordBase := TO_DINT(AxisReference - 1) * 23;
	cleanupStart := Ds402HomeState[119]$UDINT;
	cleanupExpired := (cleanupStart <> 0) & (stage >= 90) & (stage <= 99) &
		((serviceNow - cleanupStart) >= 1000);
	if cleanupExpired then
		if Ds402HomeState[94] <> 0 then
			orphanResult := -1;
			case axisReference of
				1:
					if IsClientConnected(#SdoAxis1) then
						orphanResult := SdoAxis1.MarkOrphan(Ds402HomeState[99]$UDINT);
					end_if;
				2:
					if IsClientConnected(#SdoAxis2) then
						orphanResult := SdoAxis2.MarkOrphan(Ds402HomeState[99]$UDINT);
					end_if;
				3:
					if IsClientConnected(#SdoAxis3) then
						orphanResult := SdoAxis3.MarkOrphan(Ds402HomeState[99]$UDINT);
					end_if;
				4:
					if IsClientConnected(#SdoAxis4) then
						orphanResult := SdoAxis4.MarkOrphan(Ds402HomeState[99]$UDINT);
					end_if;
			end_case;
			// MarkOrphan acceptance is not executor retirement proof. Keep every
			// pending flag and retain exact-token uncertainty in quarantine.
			Ds402HomeState[127] := 1;
		end_if;
		if Ds402HomeState[113] <> 0 then
			Ds402HomeState[127] := 1;
		end_if;
		ownerResult := -1;
		if IsClientConnected(#AxisOwnership) then
			if preemptionCleanup then
				ownerResult :=
					AxisOwnership.PublishAxisOwnershipPreemptionCleanup(
						ExpectedAxisMask:=axisMask,
						PreemptedAdmissionToken:=admissionToken,
						PreemptedOwnerGeneration:=ownerGeneration,
						SafetyAdmissionToken:=safetyAdmissionToken,
						SafetyOwnerGeneration:=safetyOwnerGeneration,
						CleanupKind:=
							LMC_DIAG_PREEMPT_CLEANUP_INCOMPLETE_QUARANTINE,
						ReportValue0:=Ds402HomeState[107]$UDINT,
						ReportValue1:=Ds402HomeState[108]$UDINT,
						ObservationCycle:=currentCycle);
				if (ownerResult <> 0) & (ownerResult <> 1) then
					Ds402HomeState[119] := ownerResult;
					Ds402HomeState[118]$UDINT :=
						LMC_DIAG_DS402_PUBLISH_FAILURE_MAGIC;
					Ds402HomeState[92] := 101;
					RETURN;
				end_if;
			else
				ownerResult := AxisOwnership.PublishAxisOwnership(
					AxisMask:=axisMask,
					AdmissionToken:=admissionToken,
					OwnerGeneration:=ownerGeneration,
					ReportKind:=LMC_DIAG_OWNER_REPORT_QUARANTINE,
					ReportValue0:=Ds402HomeState[107]$UDINT,
					ReportValue1:=Ds402HomeState[108]$UDINT,
					ObservationCycle:=currentCycle);
				if ownerResult <> 0 then
					Ds402HomeState[119] := ownerResult;
					Ds402HomeState[118]$UDINT :=
						LMC_DIAG_DS402_PUBLISH_FAILURE_MAGIC;
					Ds402HomeState[92] := 101;
					RETURN;
				end_if;
			end_if;
		else
			Ds402HomeState[119] := ownerResult;
			Ds402HomeState[118]$UDINT :=
				LMC_DIAG_DS402_PUBLISH_FAILURE_MAGIC;
			Ds402HomeState[92] := 101;
			RETURN;
		end_if;
		Ds402HomeState[92] := 101;
		RETURN;
	end_if;

	case stage of
		90:
			if IsClientConnected(#InputLatch) then
				mailboxResult := InputLatch.RequestDs402HomeSafetyDrain(
					OperationToken:=Ds402HomeState[101]$UDINT,
					AxisReference:=axisReference);
				if mailboxResult = 0 then
					Ds402HomeState[117] := 0;
					Ds402HomeState[92] := 92;
				elsif mailboxResult <> 1 then
					// Stay in bounded cleanup until timeout; never infer LOW.
					Ds402HomeState[108] := TO_DINT(0 - mailboxResult);
				end_if;
			end_if;
		91:
			// Recover an older cleanup stage through the durable drain path.
			Ds402HomeState[92] := 90;
		92:
			if Ds402HomeState[116] = 0 then
				// Stage 94 also drains a timeout-raced SDO before any terminal record.
				Ds402HomeState[92] := 94;
			elsif Ds402HomeState[104] = 0 then
				Ds402HomeState[92] := 94;
			elsif IsClientConnected(#InputLatch) then
				mailboxResult := InputLatch.SubmitDs402HomeSetpointAlignment(
					Ds402HomeState[101]$UDINT, axisReference, actualPosition);
				if mailboxResult = 0 then
					Ds402HomeState[92] := 94;
				elsif mailboxResult = 1 then
					Ds402HomeState[92] := 93;
				else
					Ds402HomeState[108] := TO_DINT(0 - mailboxResult);
					Ds402HomeState[92] := 98;
				end_if;
			end_if;
		93:
			if IsClientConnected(#InputLatch) then
				mailboxResult := InputLatch.GetDs402HomeControlState(
					Ds402HomeState[101]$UDINT);
				if mailboxResult = 0 then
					Ds402HomeState[92] := 94;
				elsif mailboxResult <> 1 then
					Ds402HomeState[108] := TO_DINT(0 - mailboxResult);
					Ds402HomeState[92] := 98;
				end_if;
			end_if;
		94:
			// MarkOrphan returns -2 when completion may already be ready. Drain
			// that exact token before waiting for IsReusable and restoring CSP.
			if Ds402HomeState[113] <> 0 then
				completionResult := -2;
				case axisReference of
					1:
						if IsClientConnected(#SdoAxis1) then
							completionResult := SdoAxis1.CopyCompletion(
								Ds402HomeState[99]$UDINT, #completion,
								sizeof(completion));
						end_if;
					2:
						if IsClientConnected(#SdoAxis2) then
							completionResult := SdoAxis2.CopyCompletion(
								Ds402HomeState[99]$UDINT, #completion,
								sizeof(completion));
						end_if;
					3:
						if IsClientConnected(#SdoAxis3) then
							completionResult := SdoAxis3.CopyCompletion(
								Ds402HomeState[99]$UDINT, #completion,
								sizeof(completion));
						end_if;
					4:
						if IsClientConnected(#SdoAxis4) then
							completionResult := SdoAxis4.CopyCompletion(
								Ds402HomeState[99]$UDINT, #completion,
								sizeof(completion));
						end_if;
				end_case;
				if completionResult = 0 then
					Ds402HomeState[94] := 0;
					Ds402HomeState[113] := 0;
					Ds402HomeState[127] := 0;
				end_if;
			end_if;
			executorConnected := FALSE;
			executorReusable := FALSE;
			case axisReference of
				1:
					executorConnected := IsClientConnected(#SdoAxis1) <> 0;
					if executorConnected then
						executorReusable := SdoAxis1.IsReusable();
					end_if;
				2:
					executorConnected := IsClientConnected(#SdoAxis2) <> 0;
					if executorConnected then
						executorReusable := SdoAxis2.IsReusable();
					end_if;
				3:
					executorConnected := IsClientConnected(#SdoAxis3) <> 0;
					if executorConnected then
						executorReusable := SdoAxis3.IsReusable();
					end_if;
				4:
					executorConnected := IsClientConnected(#SdoAxis4) <> 0;
					if executorConnected then
						executorReusable := SdoAxis4.IsReusable();
					end_if;
			end_case;
			if executorConnected = FALSE then
				Ds402HomeState[92] := 98;
			elsif executorReusable then
				Ds402HomeState[113] := 0;
				if Ds402HomeState[116] = 0 then
					Ds402HomeState[92] := 98;
				else
					ownerResult := -3;
					if preemptionCleanup then
						// The coordinator snapshot authorizes only this cleanup SDO.
						ownerResult := 0;
					end_if;
					if IsClientConnected(#AxisOwnership) &
						(preemptionCleanup = FALSE) then
						ownerResult := AxisOwnership.ValidateAxisOwnership(
							CommandId:=0x7D15,
							Reference:=axisReference,
							ExpectedAxisMask:=axisMask,
							OwnerKind:=LMC_DIAG_OWNER_KIND_DS402_HOME,
							ResourceKind:=LMC_DIAG_RESOURCE_DS402_HOME,
							AdmissionMode:=LMC_DIAG_ADMISSION_LIFECYCLE,
							CallerSessionEpoch:=ds402ProcessOwnerSessionEpoch,
							RequestSequence:=ownerRequestSequence,
							AdmissionToken:=admissionToken,
							OwnerGeneration:=ownerGeneration,
							RequiredPhase:=LMC_DIAG_OWNER_PHASE_ACTIVE);
					end_if;
					if ownerResult <> 0 then
						Ds402HomeState[108] := TO_DINT(0 - ownerResult);
						Ds402HomeState[92] := 98;
					else
						sdoToken := Ds402HomeState[99]$UDINT + 1;
						if sdoToken = 0 then
							sdoToken := 1;
						end_if;
						Ds402HomeState[99] := sdoToken$DINT;
						sdoData := 8;
						startResult := ERROR;
						case axisReference of
							1: startResult := SdoAxis1.TryStartWrite(sdoToken, 0x6060, 0, (#sdoData)$^USINT, 1, 1000);
							2: startResult := SdoAxis2.TryStartWrite(sdoToken, 0x6060, 0, (#sdoData)$^USINT, 1, 1000);
							3: startResult := SdoAxis3.TryStartWrite(sdoToken, 0x6060, 0, (#sdoData)$^USINT, 1, 1000);
							4: startResult := SdoAxis4.TryStartWrite(sdoToken, 0x6060, 0, (#sdoData)$^USINT, 1, 1000);
						end_case;
						if startResult = READY then
							Ds402HomeState[112] := currentCycle$DINT;
							Ds402HomeState[94] := 1;
							Ds402HomeState[92] := 95;
						elsif startResult = ERROR then
							Ds402HomeState[92] := 98;
						end_if;
					end_if;
				end_if;
			end_if;
		95:
			completionResult := -2;
			case axisReference of
				1:
					if IsClientConnected(#SdoAxis1) then
						completionResult := SdoAxis1.CopyCompletion(
							Ds402HomeState[99]$UDINT, #completion, sizeof(completion));
					end_if;
				2:
					if IsClientConnected(#SdoAxis2) then
						completionResult := SdoAxis2.CopyCompletion(
							Ds402HomeState[99]$UDINT, #completion, sizeof(completion));
					end_if;
				3:
					if IsClientConnected(#SdoAxis3) then
						completionResult := SdoAxis3.CopyCompletion(
							Ds402HomeState[99]$UDINT, #completion, sizeof(completion));
					end_if;
				4:
					if IsClientConnected(#SdoAxis4) then
						completionResult := SdoAxis4.CopyCompletion(
							Ds402HomeState[99]$UDINT, #completion, sizeof(completion));
					end_if;
			end_case;
			if completionResult = 0 then
				Ds402HomeState[94] := 0;
				if (completion.ValidationCode = 0) & (completion.OsResult = 0) &
					(completion.AbortCode = 0) & (completion.ObjectIndex = 0x6060) &
					(completion.IsWrite <> 0) & (completion.ActualLength = 1) then
					Ds402HomeState[92] := 96;
				else
					Ds402HomeState[92] := 98;
				end_if;
			elsif (completionResult <> -2) & (completionResult <> -3) then
				// Token mismatch or executor quarantine is not retirement proof.
				Ds402HomeState[127] := 1;
				Ds402HomeState[92] := 98;
			end_if;
		96:
			executorReusable := FALSE;
			case axisReference of
				1:
					if IsClientConnected(#SdoAxis1) then
						executorReusable := SdoAxis1.IsReusable();
					end_if;
				2:
					if IsClientConnected(#SdoAxis2) then
						executorReusable := SdoAxis2.IsReusable();
					end_if;
				3:
					if IsClientConnected(#SdoAxis3) then
						executorReusable := SdoAxis3.IsReusable();
					end_if;
				4:
					if IsClientConnected(#SdoAxis4) then
						executorReusable := SdoAxis4.IsReusable();
					end_if;
			end_case;
			if executorReusable then
				ownerResult := -3;
				if preemptionCleanup then
					// The old active tuple is intentionally hidden by safety overlay.
					ownerResult := 0;
				end_if;
				if IsClientConnected(#AxisOwnership) &
					(preemptionCleanup = FALSE) then
					ownerResult := AxisOwnership.ValidateAxisOwnership(
						CommandId:=0x7D15,
						Reference:=axisReference,
						ExpectedAxisMask:=axisMask,
						OwnerKind:=LMC_DIAG_OWNER_KIND_DS402_HOME,
						ResourceKind:=LMC_DIAG_RESOURCE_DS402_HOME,
						AdmissionMode:=LMC_DIAG_ADMISSION_LIFECYCLE,
						CallerSessionEpoch:=ds402ProcessOwnerSessionEpoch,
						RequestSequence:=ownerRequestSequence,
						AdmissionToken:=admissionToken,
						OwnerGeneration:=ownerGeneration,
						RequiredPhase:=LMC_DIAG_OWNER_PHASE_ACTIVE);
				end_if;
				if ownerResult <> 0 then
					Ds402HomeState[108] := TO_DINT(0 - ownerResult);
					Ds402HomeState[92] := 98;
				else
					sdoToken := Ds402HomeState[99]$UDINT + 1;
					if sdoToken = 0 then
						sdoToken := 1;
					end_if;
					Ds402HomeState[99] := sdoToken$DINT;
					startResult := ERROR;
					case axisReference of
						1: startResult := SdoAxis1.TryStartRead(sdoToken, 0x6061, 0, 1, 1000);
						2: startResult := SdoAxis2.TryStartRead(sdoToken, 0x6061, 0, 1, 1000);
						3: startResult := SdoAxis3.TryStartRead(sdoToken, 0x6061, 0, 1, 1000);
						4: startResult := SdoAxis4.TryStartRead(sdoToken, 0x6061, 0, 1, 1000);
					end_case;
					if startResult = READY then
						Ds402HomeState[112] := currentCycle$DINT;
						Ds402HomeState[94] := 1;
						Ds402HomeState[92] := 97;
					elsif startResult = ERROR then
						Ds402HomeState[92] := 98;
					end_if;
				end_if;
			end_if;
		97:
			completionResult := -2;
			case axisReference of
				1:
					if IsClientConnected(#SdoAxis1) then
						completionResult := SdoAxis1.CopyCompletion(
							Ds402HomeState[99]$UDINT, #completion, sizeof(completion));
					end_if;
				2:
					if IsClientConnected(#SdoAxis2) then
						completionResult := SdoAxis2.CopyCompletion(
							Ds402HomeState[99]$UDINT, #completion, sizeof(completion));
					end_if;
				3:
					if IsClientConnected(#SdoAxis3) then
						completionResult := SdoAxis3.CopyCompletion(
							Ds402HomeState[99]$UDINT, #completion, sizeof(completion));
					end_if;
				4:
					if IsClientConnected(#SdoAxis4) then
						completionResult := SdoAxis4.CopyCompletion(
							Ds402HomeState[99]$UDINT, #completion, sizeof(completion));
					end_if;
			end_case;
			if completionResult = 0 then
				Ds402HomeState[94] := 0;
				if (completion.ValidationCode = 0) & (completion.OsResult = 0) &
					(completion.AbortCode = 0) & (completion.ObjectIndex = 0x6061) &
					(completion.IsWrite = 0) & (completion.ActualLength = 1) &
					((completion.Data and 0xFF) = 8) then
					Ds402HomeState[116] := 0;
				end_if;
				Ds402HomeState[92] := 98;
			elsif (completionResult <> -2) & (completionResult <> -3) then
				// Preserve the pending tuple and force incomplete quarantine.
				Ds402HomeState[127] := 1;
				Ds402HomeState[92] := 98;
			end_if;
		98:
			if Ds402HomeState[117] = 0 then
				Ds402HomeState[92] := 100;
			else
				Ds402HomeState[92] := 90;
			end_if;
		99:
			Ds402HomeState[92] := 90;
		100:
			if preemptionCleanup then
				// SAFE requires bit 4 low, CSP readback, RT release and an idle
				// exact SDO executor. Every weaker outcome stays quarantined.
				executorConnected := FALSE;
				executorReusable := FALSE;
				case axisReference of
					1:
						executorConnected := IsClientConnected(#SdoAxis1) <> 0;
						if executorConnected then
							executorReusable := SdoAxis1.IsReusable();
						end_if;
					2:
						executorConnected := IsClientConnected(#SdoAxis2) <> 0;
						if executorConnected then
							executorReusable := SdoAxis2.IsReusable();
						end_if;
					3:
						executorConnected := IsClientConnected(#SdoAxis3) <> 0;
						if executorConnected then
							executorReusable := SdoAxis3.IsReusable();
						end_if;
					4:
						executorConnected := IsClientConnected(#SdoAxis4) <> 0;
						if executorConnected then
							executorReusable := SdoAxis4.IsReusable();
						end_if;
				end_case;
				preemptionCleanupKind :=
					LMC_DIAG_PREEMPT_CLEANUP_INCOMPLETE_QUARANTINE;
				if (Ds402HomeState[117] = 0) &
					(Ds402HomeState[94] = 0) &
					(Ds402HomeState[113] = 0) &
					(Ds402HomeState[116] = 0) &
					(Ds402HomeState[127] = 0) &
					executorConnected & executorReusable then
					preemptionCleanupKind :=
						LMC_DIAG_PREEMPT_CLEANUP_SAFE;
				end_if;
				ownerResult :=
					AxisOwnership.PublishAxisOwnershipPreemptionCleanup(
						ExpectedAxisMask:=axisMask,
						PreemptedAdmissionToken:=admissionToken,
						PreemptedOwnerGeneration:=ownerGeneration,
						SafetyAdmissionToken:=safetyAdmissionToken,
						SafetyOwnerGeneration:=safetyOwnerGeneration,
						CleanupKind:=preemptionCleanupKind,
						ReportValue0:=Ds402HomeState[107]$UDINT,
						ReportValue1:=Ds402HomeState[108]$UDINT,
						ObservationCycle:=currentCycle);
				if (ownerResult <> 0) & (ownerResult <> 1) then
					Ds402HomeState[119] := ownerResult;
					Ds402HomeState[118]$UDINT :=
						LMC_DIAG_DS402_PUBLISH_FAILURE_MAGIC;
					Ds402HomeState[92] := 101;
					RETURN;
				end_if;
				if preemptionCleanupKind =
					LMC_DIAG_PREEMPT_CLEANUP_SAFE then
					if currentCycle <
						Ds402HomeState[recordBase + 19]$UDINT then
						currentCycle :=
							Ds402HomeState[recordBase + 19]$UDINT;
					end_if;
					Ds402HomeState[recordBase + 14] := 1;
					Ds402HomeState[recordBase + 15] :=
						LMC_DIAG_ADMIN_ERROR_ID;
					Ds402HomeState[recordBase + 16] := 31;
					Ds402HomeState[recordBase + 20] := currentCycle$DINT;
					Ds402HomeState[recordBase + 21] := 0;
					Ds402HomeState[101] := 0;
					Ds402HomeState[recordBase] := 4;
					Ds402HomeState[92] := 0;
				else
					Ds402HomeState[92] := 101;
				end_if;
				RETURN;
			elsif Ds402HomeState[117] <> 0 then
				// Never publish a terminal record while RT ownership is uncertain.
				Ds402HomeState[92] := 99;
			elsif (Ds402HomeState[94] <> 0) |
				(Ds402HomeState[113] <> 0) |
				(Ds402HomeState[116] <> 0) |
				(Ds402HomeState[127] <> 0) then
				// A non-reusable executor or unverified CSP mode is quarantined.
				Ds402HomeState[92] := 101;
			else
				ownerResult := -1;
				if Ds402HomeState[126] = 0 then
					if currentCycle <
						Ds402HomeState[recordBase + 19]$UDINT then
						currentCycle :=
							Ds402HomeState[recordBase + 19]$UDINT;
					end_if;
					Ds402HomeState[106] := 3;
					Ds402HomeState[recordBase + 14] := 1;
					if Ds402HomeState[107] = 11 then
						Ds402HomeState[recordBase + 15] := -6;
					else
						Ds402HomeState[recordBase + 15] :=
							LMC_DIAG_ADMIN_ERROR_ID;
					end_if;
					Ds402HomeState[recordBase + 16] :=
						Ds402HomeState[107];
					Ds402HomeState[recordBase + 20] := currentCycle$DINT;
					Ds402HomeState[recordBase + 21] :=
						Ds402HomeState[108];
					if IsClientConnected(#AxisOwnership) then
						ownerResult :=
							AxisOwnership.PublishAxisOwnershipDs402Receipt(
								AxisMask:=axisMask,
								AdmissionToken:=admissionToken,
								OwnerGeneration:=ownerGeneration,
								ReportKind:=
									LMC_DIAG_OWNER_REPORT_TERMINAL_SAFE_FAILURE,
								ReportValue0:=Ds402HomeState[107]$UDINT,
								ReportValue1:=Ds402HomeState[108]$UDINT,
								ObservationCycle:=currentCycle,
								pDs402State:=#Ds402HomeState[0],
								Ds402StateSize:=sizeof(Ds402HomeState));
					end_if;
					if ownerResult = 0 then
						Ds402HomeState[125] := 2;
						ownerResult :=
							AxisOwnership.PublishAxisOwnershipDs402Receipt(
								AxisMask:=axisMask,
								AdmissionToken:=admissionToken,
								OwnerGeneration:=ownerGeneration,
								ReportKind:=
									LMC_DIAG_OWNER_REPORT_TERMINAL_SAFE_FAILURE,
								ReportValue0:=Ds402HomeState[107]$UDINT,
								ReportValue1:=Ds402HomeState[108]$UDINT,
								ObservationCycle:=currentCycle,
								pDs402State:=#Ds402HomeState[0],
								Ds402StateSize:=sizeof(Ds402HomeState));
						if ownerResult = 1 then
							Ds402HomeState[92] :=
								LMC_DIAG_DS402_STAGE_FINALIZE;
						elsif ownerResult <> 0 then
							Ds402HomeState[92] := 101;
						end_if;
						RETURN;
					elsif ownerResult = 1 then
						Ds402HomeState[92] :=
							LMC_DIAG_DS402_STAGE_FINALIZE;
						RETURN;
					else
						Ds402HomeState[92] := 101;
					end_if;
				else
					ownerResult := -1;
					if IsClientConnected(#AxisOwnership) then
						// Once an SDO dispatch was reported, a non-success path
						// remains quarantined instead of claiming safe release.
						ownerResult := AxisOwnership.PublishAxisOwnership(
							AxisMask:=axisMask,
							AdmissionToken:=admissionToken,
							OwnerGeneration:=ownerGeneration,
							ReportKind:=LMC_DIAG_OWNER_REPORT_QUARANTINE,
							ReportValue0:=Ds402HomeState[107]$UDINT,
							ReportValue1:=Ds402HomeState[108]$UDINT,
							ObservationCycle:=currentCycle);
						if ownerResult <> 0 then
							Ds402HomeState[119] := ownerResult;
							Ds402HomeState[118]$UDINT :=
								LMC_DIAG_DS402_PUBLISH_FAILURE_MAGIC;
							Ds402HomeState[92] := 101;
							RETURN;
						end_if;
					else
						Ds402HomeState[119] := ownerResult;
						Ds402HomeState[118]$UDINT :=
							LMC_DIAG_DS402_PUBLISH_FAILURE_MAGIC;
						Ds402HomeState[92] := 101;
						RETURN;
					end_if;
				end_if;
				if Ds402HomeState[126] <> 0 then
					Ds402HomeState[92] := 101;
				end_if;
			end_if;
		101:
			// Fail-closed quarantine. A PLC restart or a future explicit recovery
			// command is required; generic D5 remains excluded while stage is nonzero.
			RETURN;
	end_case;

END_FUNCTION

FUNCTION LMCDiagnosticsService::HandleDiagnosticsCapabilities
	VAR_INPUT
		RequestSize 	: UDINT;
		pResponse 	: ^USINT;
		ResponseCapacity 	: UDINT;
		CurrentDiagnosticsBootId 	: UDINT;
		DetailCode 	: UDINT;
	END_VAR
	VAR_OUTPUT
		ResponseSize 	: DINT;
	END_VAR
	VAR
		localDetailCode : UDINT;
	END_VAR

	ResponseSize := -1;
	if (pResponse = NIL) | (ResponseCapacity < 68) then
		RETURN;
	end_if;

	localDetailCode := DetailCode;
	if RequestSize <> 8 then
		localDetailCode := 12;
	end_if;
	if localDetailCode <> 0 then
		(pResponse + 4)^$UINT := 1;
		(pResponse + 6)^$INT := LMC_DIAG_ERROR_ID;
		(pResponse + 12)^$UDINT := localDetailCode;
	end_if;
	(pResponse + 16)^$UDINT := 1;
	(pResponse + 20)^$UDINT := 0x00004007;
	(pResponse + 24)^$UDINT := LMC_DIAG_MAP_REVISION;
	(pResponse + 28)^$UINT := 24;
	(pResponse + 30)^$UINT := 0;
	(pResponse + 32)^$UINT := 0;
	(pResponse + 34)^$UINT := 0;
	(pResponse + 36)^$UDINT := 0;
	(pResponse + 40)^$UDINT := 1000;
	(pResponse + 44)^$UINT := 1320;
	(pResponse + 46)^$UINT := 2040;
	(pResponse + 48)^$UINT := 1280;
	(pResponse + 50)^$UINT := 80;
	(pResponse + 52)^$UINT := 16;
	(pResponse + 54)^$UINT := 0;
	(pResponse + 56)^$UDINT := 0;
	(pResponse + 60)^$UINT := 0;
	(pResponse + 62)^$UINT := 0;
	(pResponse + 64)^$UDINT := CurrentDiagnosticsBootId;
	if CurrentDiagnosticsBootId <> 0 then
		(pResponse + 20)^$UDINT := 0x0000613F;
		(pResponse + 30)^$UINT := 24;
		(pResponse + 32)^$UINT := 24;
		(pResponse + 34)^$UINT := 1;
		(pResponse + 36)^$UDINT := 320000;
		(pResponse + 56)^$UDINT := 1280000;
		(pResponse + 60)^$UINT := 4;
		if (LMC_DIAG_D5_SDO_WRITE_GLOBAL_ENABLED = TRUE) &
			((LMC_DIAG_D5_SDO_WRITE_UI24_AXIS1_ENABLED = TRUE) |
			 (LMC_DIAG_D5_SDO_WRITE_UI24_AXIS2_ENABLED = TRUE) |
			 (LMC_DIAG_D5_SDO_WRITE_UI24_AXIS3_ENABLED = TRUE) |
			 (LMC_DIAG_D5_SDO_WRITE_UI24_AXIS4_ENABLED = TRUE)) then
			(pResponse + 20)^$UDINT :=
				(pResponse + 20)^$UDINT OR 0x00000200;
		end_if;
		if LMC_DIAG_ENCODER_TW20_ENABLED = TRUE then
			(pResponse + 20)^$UDINT :=
				(pResponse + 20)^$UDINT OR 0x00040000;
		end_if;
		if LMC_DIAG_ENCODER_TW19_ENABLED = TRUE then
			(pResponse + 20)^$UDINT :=
				(pResponse + 20)^$UDINT OR 0x00080000;
		end_if;
	end_if;
	ResponseSize := 68;

END_FUNCTION

FUNCTION LMCDiagnosticsService::HandleDiagnosticsBulkRequest
	VAR_INPUT
		CommandId 	: UINT;
		pRequest 	: ^USINT;
		RequestSize 	: UDINT;
		pResponse 	: ^USINT;
		ResponseCapacity 	: UDINT;
		CallerSessionEpoch 	: UDINT;
	END_VAR
	VAR_OUTPUT
		ResponseSize 	: DINT;
	END_VAR
	VAR
		physicalAxis, signalCode, catalogIndex, signalCount : UINT;
		duplicateIndex, entryIndex : UINT;
		expectedMapRevision, requestedBulkId, signalId : UDINT;
		expectedRequestSize, requestBulkId, requestConfigRevision : UDINT;
		healthOffset, valueOffset, entryOffset, entryDetailCode : UDINT;
		detailCode : UDINT;
		valueType, entryStatus : USINT;
		copyResult : DINT;
		snapshot : ARRAY [0..303] OF USINT;
		hasInvalidEntry : BOOL;
	END_VAR

	ResponseSize := -1;
	detailCode := 0;

	case CommandId of
		0x7E30:
			if RequestSize < 20 then
				detailCode := 12;
			else
				expectedMapRevision := (pRequest + 8)^$UDINT;
				requestedBulkId := (pRequest + 12)^$UDINT;
				signalCount := (pRequest + 16)^$UINT;
				expectedRequestSize := 20 + TO_UDINT(signalCount) * 4;
				if expectedMapRevision <> LMC_DIAG_MAP_REVISION then
					detailCode := 3;
				elsif (CallerSessionEpoch = 0) | (signalCount = 0) |
					(signalCount > LMC_DIAG_MAX_BULK_SIGNALS) |
					((pRequest + 18)^$UINT <> 0) |
					(RequestSize <> expectedRequestSize) then
					detailCode := 12;
				elsif ResponseCapacity < 36 then
					detailCode := 20;
				end_if;

				if detailCode = 0 then
					for entryIndex := 0 to signalCount - 1 do
						signalId := (pRequest + 20 + TO_UDINT(entryIndex) * 4)^$UDINT;
						physicalAxis := TO_UINT((signalId shr 8) and 0xFF);
						signalCode := TO_UINT(signalId and 0xFF);
						if (physicalAxis < 1) | (physicalAxis > 4) |
							(signalCode < 1) | (signalCode > 6) |
							(signalId <> (0x00100000 or
							 (TO_UDINT(physicalAxis) shl 8) or TO_UDINT(signalCode))) then
							detailCode := 4;
						elsif entryIndex > 0 then
							for duplicateIndex := 0 to entryIndex - 1 do
								if signalId =
									(pRequest + 20 + TO_UDINT(duplicateIndex) * 4)^$UDINT then
									detailCode := 12;
								end_if;
							end_for;
						end_if;
					end_for;
				end_if;

				if (detailCode = 0) & (BulkState <> 0) &
					(BulkOwnerSessionEpoch <> CallerSessionEpoch) then
					BulkId := 0;
					BulkConfigRevision := 0;
					BulkOwnerSessionEpoch := 0;
					BulkConfiguredCycle := 0;
					BulkActivationCycle := 0;
					BulkState := 0;
					BulkSignalCount := 0;
					_memset(dest:=#BulkSignalIds[0], usByte:=0,
						cntr:=sizeof(BulkSignalIds));
				end_if;

				if (detailCode = 0) & (BulkState <> 0) then
					if requestedBulkId = 0 then
						detailCode := 9;
					elsif requestedBulkId <> BulkId then
						detailCode := 10;
					end_if;
				end_if;
				if (detailCode = 0) &
					((NextBulkConfigRevision = 0xFFFFFFFF) |
					 ((BulkState = 0) & (requestedBulkId = 0) &
					  (NextBulkId = 0xFFFFFFFF))) then
					detailCode := 19;
				end_if;

				if detailCode = 0 then
					if IsClientConnected(#InputLatch) = FALSE then
						detailCode := 11;
					else
						copyResult := InputLatch.CopySnapshot(
							pDest:=#snapshot[0], DestSize:=sizeof(snapshot));
						if copyResult <> 0 then
							detailCode := 9;
						end_if;
					end_if;
				end_if;

				if detailCode = 0 then
					if BulkState = 0 then
						if requestedBulkId = 0 then
							NextBulkId += 1;
							BulkId := NextBulkId;
						else
							BulkId := requestedBulkId;
						end_if;
					end_if;

					NextBulkConfigRevision += 1;
					BulkConfigRevision := NextBulkConfigRevision;
					BulkOwnerSessionEpoch := CallerSessionEpoch;
					BulkConfiguredCycle := snapshot[0]$UDINT;
					BulkActivationCycle := 0;
					BulkState := 1;
					BulkSignalCount := signalCount;
					_memset(dest:=#BulkSignalIds[0], usByte:=0,
						cntr:=sizeof(BulkSignalIds));
					for entryIndex := 0 to signalCount - 1 do
						BulkSignalIds[entryIndex] :=
							(pRequest + 20 + TO_UDINT(entryIndex) * 4)^$UDINT;
					end_for;

					(pResponse + 16)^$UDINT := BulkId;
					(pResponse + 20)^$UDINT := BulkConfigRevision;
					(pResponse + 24)^$UDINT := LMC_DIAG_MAP_REVISION;
					(pResponse + 28)^$UINT := BulkState;
					(pResponse + 30)^$UINT := BulkSignalCount;
					(pResponse + 32)^$UDINT := BulkActivationCycle;
					ResponseSize := 36;
				end_if;
			end_if;

		0x7E31:
			if RequestSize <> 20 then
				detailCode := 12;
			else
				requestBulkId := (pRequest + 8)^$UDINT;
				requestConfigRevision := (pRequest + 12)^$UDINT;
				expectedMapRevision := (pRequest + 16)^$UDINT;
				if expectedMapRevision <> LMC_DIAG_MAP_REVISION then
					detailCode := 3;
				elsif (requestBulkId = 0) | (requestConfigRevision = 0) then
					detailCode := 12;
				elsif (BulkState = 0) | (requestBulkId <> BulkId) |
					(requestConfigRevision <> BulkConfigRevision) |
					(CallerSessionEpoch <> BulkOwnerSessionEpoch) then
					detailCode := 10;
				elsif IsClientConnected(#InputLatch) = FALSE then
					detailCode := 11;
				else
					copyResult := InputLatch.CopySnapshot(
						pDest:=#snapshot[0], DestSize:=sizeof(snapshot));
					if copyResult <> 0 then
						detailCode := 9;
					elsif (BulkState = 1) &
						(snapshot[0]$UDINT <> BulkConfiguredCycle) then
						BulkState := 2;
						BulkActivationCycle := snapshot[0]$UDINT;
					end_if;
				end_if;

				if detailCode = 0 then
					if ResponseCapacity < 36 then
						detailCode := 20;
					else
						(pResponse + 16)^$UDINT := BulkId;
						(pResponse + 20)^$UDINT := BulkConfigRevision;
						(pResponse + 24)^$UDINT := LMC_DIAG_MAP_REVISION;
						(pResponse + 28)^$UINT := BulkState;
						(pResponse + 30)^$UINT := BulkSignalCount;
						(pResponse + 32)^$UDINT := BulkActivationCycle;
						ResponseSize := 36;
					end_if;
				end_if;
			end_if;

		0x7E32:
			if RequestSize <> 20 then
				detailCode := 12;
			else
				requestBulkId := (pRequest + 8)^$UDINT;
				requestConfigRevision := (pRequest + 12)^$UDINT;
				expectedMapRevision := (pRequest + 16)^$UDINT;
				if expectedMapRevision <> LMC_DIAG_MAP_REVISION then
					detailCode := 3;
				elsif (requestBulkId = 0) | (requestConfigRevision = 0) then
					detailCode := 12;
				elsif (BulkState = 0) | (requestBulkId <> BulkId) |
					(requestConfigRevision <> BulkConfigRevision) |
					(CallerSessionEpoch <> BulkOwnerSessionEpoch) then
					detailCode := 10;
				elsif IsClientConnected(#InputLatch) = FALSE then
					detailCode := 11;
				else
					copyResult := InputLatch.CopySnapshot(
						pDest:=#snapshot[0], DestSize:=sizeof(snapshot));
					if copyResult <> 0 then
						detailCode := 9;
					elsif (BulkState = 1) &
						(snapshot[0]$UDINT <> BulkConfiguredCycle) then
						BulkState := 2;
						BulkActivationCycle := snapshot[0]$UDINT;
					end_if;
				end_if;

				if (detailCode = 0) & (BulkState <> 2) then
					detailCode := 11;
				end_if;
				if (detailCode = 0) &
					(ResponseCapacity < (56 + TO_UDINT(BulkSignalCount) * 16)) then
					detailCode := 20;
				end_if;

				if detailCode = 0 then
					(pResponse + 16)^$UDINT := BulkId;
					(pResponse + 20)^$UDINT := BulkConfigRevision;
					(pResponse + 24)^$UDINT := LMC_DIAG_MAP_REVISION;
					(pResponse + 28)^$UDINT := snapshot[0]$UDINT;
					(pResponse + 32)^$UDINT := snapshot[4]$UDINT;
					(pResponse + 36)^$UDINT := snapshot[8]$UDINT;
					(pResponse + 40)^$UINT := BulkSignalCount;
					(pResponse + 42)^$UINT := 16;
					(pResponse + 44)^$USINT := 1;
					(pResponse + 48)^$UDINT := snapshot[44]$UDINT;
					(pResponse + 52)^$UDINT := 3;
					hasInvalidEntry := FALSE;

					for entryIndex := 0 to BulkSignalCount - 1 do
						signalId := BulkSignalIds[entryIndex];
						physicalAxis := TO_UINT((signalId shr 8) and 0xFF);
						signalCode := TO_UINT(signalId and 0xFF);
						catalogIndex := (physicalAxis - 1) * 6 + (signalCode - 1);
						healthOffset := 64 + TO_UDINT(physicalAxis - 1) * 36;
						valueOffset := 208 + TO_UDINT(catalogIndex) * 4;
						entryOffset := 56 + TO_UDINT(entryIndex) * 16;
						valueType := 8;
						if (signalCode = 1) | (signalCode = 4) then
							valueType := 4;
						elsif (signalCode = 3) | (signalCode = 6) then
							valueType := 7;
						end_if;

						entryStatus := 0;
						if snapshot[12]$UDINT <> 8 then
							entryStatus := entryStatus or 4;
						end_if;
						if snapshot[16]$UDINT <> 0 then
							entryStatus := entryStatus or 2;
						end_if;
						if snapshot[TO_DINT(healthOffset)]$DINT = 0 then
							entryStatus := entryStatus or 8;
						end_if;
						if snapshot[TO_DINT(healthOffset + 4)]$UDINT <> 8 then
							entryStatus := entryStatus or 16;
						end_if;
						if snapshot[TO_DINT(healthOffset + 12)]$UDINT <> 0 then
							entryStatus := entryStatus or 32;
						end_if;
						if snapshot[TO_DINT(healthOffset + 16)]$UDINT = 0xFFFFFFFF then
							entryStatus := entryStatus or 128;
						end_if;

						entryDetailCode := 0;
						if entryStatus = 0 then
							entryStatus := 1;
						else
							hasInvalidEntry := TRUE;
							if (entryStatus and 8) <> 0 then
								entryDetailCode := 18;
							else
								entryDetailCode := 11;
							end_if;
						end_if;

						(pResponse + entryOffset)^$UDINT := signalId;
						(pResponse + entryOffset + 4)^$UDINT :=
							snapshot[TO_DINT(valueOffset)]$UDINT;
						(pResponse + entryOffset + 8)^$USINT := valueType;
						(pResponse + entryOffset + 9)^$USINT := entryStatus;
						(pResponse + entryOffset + 12)^$UDINT := entryDetailCode;
					end_for;

					if hasInvalidEntry then
						(pResponse + 2)^$UINT := 1;
					end_if;
					ResponseSize := 56 + TO_DINT(BulkSignalCount) * 16;
				end_if;
			end_if;

		0x7E33:
			if RequestSize <> 20 then
				detailCode := 12;
			else
				requestBulkId := (pRequest + 8)^$UDINT;
				requestConfigRevision := (pRequest + 12)^$UDINT;
				expectedMapRevision := (pRequest + 16)^$UDINT;
				if expectedMapRevision <> LMC_DIAG_MAP_REVISION then
					detailCode := 3;
				elsif (requestBulkId = 0) | (requestConfigRevision = 0) then
					detailCode := 12;
				elsif (BulkState = 0) | (requestBulkId <> BulkId) |
					(requestConfigRevision <> BulkConfigRevision) |
					(CallerSessionEpoch <> BulkOwnerSessionEpoch) then
					detailCode := 10;
				else
					BulkId := 0;
					BulkConfigRevision := 0;
					BulkOwnerSessionEpoch := 0;
					BulkConfiguredCycle := 0;
					BulkActivationCycle := 0;
					BulkState := 0;
					BulkSignalCount := 0;
					_memset(dest:=#BulkSignalIds[0], usByte:=0,
						cntr:=sizeof(BulkSignalIds));
					ResponseSize := 16;
				end_if;
			end_if;

		else
			detailCode := 2;
	end_case;

	if detailCode <> 0 then
		_memset(dest:=pResponse + 16, usByte:=0, cntr:=ResponseCapacity - 16);
		(pResponse + 2)^$UINT := 0;
		(pResponse + 4)^$UINT := 1;
		(pResponse + 6)^$INT := LMC_DIAG_ERROR_ID;
		(pResponse + 12)^$UDINT := detailCode;
		ResponseSize := 16;
	end_if;

END_FUNCTION

FUNCTION LMCDiagnosticsService::ProcessAxisOwnershipStartup
	VAR
		startupSnapshot : ARRAY [0..11] OF UDINT;
		copyResult : DINT;
		reconcileResult : DINT;
		currentBootId : UDINT;
		reportCycle : UDINT;
		drainFlags : UDINT;
		executorsReusable : BOOL;
	END_VAR

	if (IsClientConnected(#InputLatch) = FALSE) |
		(IsClientConnected(#AxisOwnership) = FALSE) then
		RETURN;
	end_if;
	copyResult := InputLatch.CopyAxisOwnershipStartupSnapshot(
		pDest:=#startupSnapshot[0], DestSize:=48);
	if copyResult <> 0 then
		RETURN;
	end_if;
	if (startupSnapshot[0] <> LMC_OWNER_STARTUP_SNAPSHOT_MAGIC) |
		(startupSnapshot[1] = 0) | (startupSnapshot[11] <> 0) then
		RETURN;
	end_if;

	drainFlags := LMC_OWNER_STARTUP_DIAG_SNAPSHOT;
	if Ds402HomeState[92] = 0 then
		drainFlags := drainFlags or LMC_OWNER_STARTUP_DIAG_DS402;
	end_if;
	if EncoderMaintenanceState[152] = 0 then
		drainFlags := drainFlags or LMC_OWNER_STARTUP_DIAG_ENCODER;
	end_if;
	if (OperationState <> LMC_DIAG_SDO_STATE_QUEUED) &
		(OperationState <> LMC_DIAG_SDO_STATE_RUNNING) &
		(SdoInternalDrainState = 0) then
		drainFlags := drainFlags or LMC_OWNER_STARTUP_DIAG_GENERIC;
	end_if;

	executorsReusable := (IsClientConnected(#SdoAxis1) <> 0) &
		(IsClientConnected(#SdoAxis2) <> 0) &
		(IsClientConnected(#SdoAxis3) <> 0) &
		(IsClientConnected(#SdoAxis4) <> 0);
	if executorsReusable then
		executorsReusable := SdoAxis1.IsReusable() & SdoAxis2.IsReusable() &
			SdoAxis3.IsReusable() & SdoAxis4.IsReusable();
	end_if;
	if executorsReusable then
		drainFlags := drainFlags or LMC_OWNER_STARTUP_DIAG_EXECUTOR;
	end_if;

	currentBootId := GetDiagnosticsBootId();
	if currentBootId = 0 then
		RETURN;
	end_if;
	reportCycle := ops.tAbsolute;
	if reportCycle = 0 then
		reportCycle := 1;
	end_if;
	reconcileResult := AxisOwnership.ReconcileAxisOwnershipStartup(
		DiagnosticsBootId:=currentBootId,
		ObservationCycle:=startupSnapshot[1],
		ReportCycle:=reportCycle,
		DiagnosticsDrainFlags:=drainFlags);

END_FUNCTION

FUNCTION GLOBAL LMCDiagnosticsService::TryTakeD5TerminalWake
	VAR_INPUT
		pTicketId 	: ^UDINT;
		pTicketBootId 	: ^UDINT;
		pOwnerSessionEpoch 	: ^UDINT;
	END_VAR
	VAR_OUTPUT
		Result 	: DINT;
	END_VAR

	Result := -1;
	if (pTicketId = NIL) | (pTicketBootId = NIL) |
		(pOwnerSessionEpoch = NIL) then
		RETURN;
	end_if;

	pTicketId^$UDINT := 0;
	pTicketBootId^$UDINT := 0;
	pOwnerSessionEpoch^$UDINT := 0;
	Result := 0;

	if (TicketId = 0) | (TicketBootId = 0) |
		(OwnerSessionEpoch = 0) then
		RETURN;
	end_if;
	if (OperationState <> LMC_DIAG_SDO_STATE_COMPLETED) &
		(OperationState <> LMC_DIAG_SDO_STATE_FAILED) &
		(OperationState <> LMC_DIAG_SDO_STATE_CANCELLED) &
		(OperationState <> LMC_DIAG_SDO_STATE_EXPIRED) then
		RETURN;
	end_if;
	if (D5TerminalWakeLastAttemptTicketId = TicketId) &
		(D5TerminalWakeLastAttemptTicketBootId = TicketBootId) &
		(D5TerminalWakeLastAttemptOwnerSessionEpoch = OwnerSessionEpoch) then
		RETURN;
	end_if;

	D5TerminalWakeLastAttemptTicketId := TicketId;
	D5TerminalWakeLastAttemptTicketBootId := TicketBootId;
	D5TerminalWakeLastAttemptOwnerSessionEpoch := OwnerSessionEpoch;
	pTicketId^$UDINT := TicketId;
	pTicketBootId^$UDINT := TicketBootId;
	pOwnerSessionEpoch^$UDINT := OwnerSessionEpoch;
	Result := 1;

END_FUNCTION

FUNCTION LMCDiagnosticsService::HandleAxisSetOperationModeStart
	VAR_INPUT
		Reference 	: UINT;
		pRequest 	: ^USINT;
		pResponse 	: ^USINT;
		ResponseCapacity 	: UDINT;
		CallerSessionEpoch 	: UDINT;
		RequestSequence 	: UDINT;
		AdmissionToken 	: UDINT;
		OwnerGeneration 	: UDINT;
		RequestSize 	: UDINT;
	END_VAR
	VAR_OUTPUT
		ResponseSize 	: DINT;
	END_VAR
	VAR
		schemaVersion, requestFlags, keySchema, keyReserved : UINT;
		requestId, diagnosticsBuild, bootId, mapRevision : UDINT;
		originalRequestId, intent0, intent1, intent2, intent3 : UDINT;
		timeoutMilliseconds, operationFlags, currentBootId, detailCode : UDINT;
		requestedMode : SINT;
		axisReference : UINT;
		reservedByte : USINT;
	END_VAR

	ResponseSize := -1;
	if (pResponse = NIL) | (ResponseCapacity < 16) then
		RETURN;
	end_if;
	_memset(dest:=pResponse, usByte:=0, cntr:=24);
	pResponse^$UINT := LMC_DIAG_SCHEMA_VERSION;
	(pResponse + 4)^$UINT := 1;
	(pResponse + 6)^$INT := LMC_DIAG_ADMIN_ERROR_ID;
	detailCode := 5;
	requestId := 0;
	requestedMode := 0;
	if (pRequest <> NIL) & (RequestSize >= 8) then
		requestId := (pRequest + 4)^$UDINT;
	end_if;
	(pResponse + 8)^$UDINT := requestId;
	(pResponse + 12)^$UDINT := detailCode;
	ResponseSize := 16;

	if (pRequest = NIL) | (RequestSize <> 56) then
		RETURN;
	end_if;
	schemaVersion := pRequest^$UINT;
	requestFlags := (pRequest + 2)^$UINT;
	keySchema := (pRequest + 8)^$UINT;
	keyReserved := (pRequest + 10)^$UINT;
	diagnosticsBuild := (pRequest + 12)^$UDINT;
	bootId := (pRequest + 16)^$UDINT;
	mapRevision := (pRequest + 20)^$UDINT;
	originalRequestId := (pRequest + 24)^$UDINT;
	intent0 := (pRequest + 28)^$UDINT;
	intent1 := (pRequest + 32)^$UDINT;
	intent2 := (pRequest + 36)^$UDINT;
	intent3 := (pRequest + 40)^$UDINT;
	axisReference := (pRequest + 44)^$UINT;
	requestedMode := (pRequest + 46)^$SINT;
	reservedByte := (pRequest + 47)^$USINT;
	timeoutMilliseconds := (pRequest + 48)^$UDINT;
	operationFlags := (pRequest + 52)^$UDINT;
	currentBootId := GetDiagnosticsBootId();

	if (schemaVersion <> 1) | (keySchema <> 1) then
		detailCode := 1;
	elsif requestFlags <> 0 then
		detailCode := 2;
	elsif requestId = 0 then
		detailCode := 3;
	elsif (Reference < 1) | (Reference > 4) |
	      (axisReference <> Reference) then
		detailCode := 4;
	elsif (keyReserved <> 0) | (reservedByte <> 0) |
	      (originalRequestId = 0) | (originalRequestId <> requestId) |
	      ((intent0 = 0) & (intent1 = 0) &
	       (intent2 = 0) & (intent3 = 0)) |
	      (timeoutMilliseconds = 0) | (operationFlags <> 0) then
		detailCode := 5;
	elsif diagnosticsBuild <> 1 then
		detailCode := 16;
	elsif (currentBootId = 0) | (bootId <> currentBootId) then
		detailCode := 17;
	elsif mapRevision <> LMC_DIAG_MAP_REVISION then
		detailCode := 18;
	elsif requestedMode <> 8 then
		detailCode := 43;
	else
		detailCode := 49;
	end_if;

	if detailCode <= 5 then
		(pResponse + 12)^$UDINT := detailCode;
		RETURN;
	end_if;
	if ResponseCapacity < 24 then
		ResponseSize := -1;
		RETURN;
	end_if;
	_memset(dest:=pResponse, usByte:=0, cntr:=24);
	pResponse^$UINT := LMC_DIAG_SCHEMA_VERSION;
	(pResponse + 4)^$UINT := 1;
	(pResponse + 6)^$INT := LMC_DIAG_ADMIN_ERROR_ID;
	(pResponse + 8)^$UDINT := requestId;
	(pResponse + 12)^$UDINT := detailCode;
	(pResponse + 16)^$DINT := TO_DINT(requestedMode);
	(pResponse + 20)^$UDINT := 0;
	ResponseSize := 24;

END_FUNCTION

FUNCTION LMCDiagnosticsService::HandleAxisSetOperationModeOutcome
	VAR_INPUT
		Reference 	: UINT;
		pRequest 	: ^USINT;
		pResponse 	: ^USINT;
		ResponseCapacity 	: UDINT;
		CallerSessionEpoch 	: UDINT;
		RequestSize 	: UDINT;
	END_VAR
	VAR_OUTPUT
		ResponseSize 	: DINT;
	END_VAR
	VAR
		schemaVersion, requestFlags, keySchema, keyReserved : UINT;
		requestId, diagnosticsBuild, bootId, mapRevision : UDINT;
		originalRequestId, intent0, intent1, intent2, intent3 : UDINT;
		timeoutMilliseconds, operationFlags, currentBootId, detailCode : UDINT;
		requestedMode : SINT;
		axisReference : UINT;
		reservedByte : USINT;
	END_VAR

	ResponseSize := -1;
	if (pResponse = NIL) | (ResponseCapacity < 16) then
		RETURN;
	end_if;
	_memset(dest:=pResponse, usByte:=0, cntr:=16);
	pResponse^$UINT := LMC_DIAG_SCHEMA_VERSION;
	(pResponse + 4)^$UINT := 1;
	(pResponse + 6)^$INT := LMC_DIAG_ADMIN_ERROR_ID;
	detailCode := 5;
	requestId := 0;
	if (pRequest <> NIL) & (RequestSize >= 8) then
		requestId := (pRequest + 4)^$UDINT;
	end_if;
	(pResponse + 8)^$UDINT := requestId;
	ResponseSize := 16;

	if (pRequest = NIL) | (RequestSize <> 56) then
		(pResponse + 12)^$UDINT := detailCode;
		RETURN;
	end_if;
	schemaVersion := pRequest^$UINT;
	requestFlags := (pRequest + 2)^$UINT;
	keySchema := (pRequest + 8)^$UINT;
	keyReserved := (pRequest + 10)^$UINT;
	diagnosticsBuild := (pRequest + 12)^$UDINT;
	bootId := (pRequest + 16)^$UDINT;
	mapRevision := (pRequest + 20)^$UDINT;
	originalRequestId := (pRequest + 24)^$UDINT;
	intent0 := (pRequest + 28)^$UDINT;
	intent1 := (pRequest + 32)^$UDINT;
	intent2 := (pRequest + 36)^$UDINT;
	intent3 := (pRequest + 40)^$UDINT;
	axisReference := (pRequest + 44)^$UINT;
	requestedMode := (pRequest + 46)^$SINT;
	reservedByte := (pRequest + 47)^$USINT;
	timeoutMilliseconds := (pRequest + 48)^$UDINT;
	operationFlags := (pRequest + 52)^$UDINT;
	currentBootId := GetDiagnosticsBootId();

	if (schemaVersion <> 1) | (keySchema <> 1) then
		detailCode := 1;
	elsif requestFlags <> 0 then
		detailCode := 2;
	elsif requestId = 0 then
		detailCode := 3;
	elsif (Reference < 1) | (Reference > 4) |
	      (axisReference <> Reference) then
		detailCode := 4;
	elsif (keyReserved <> 0) | (reservedByte <> 0) |
	      (originalRequestId = 0) |
	      ((intent0 = 0) & (intent1 = 0) &
	       (intent2 = 0) & (intent3 = 0)) |
	      (timeoutMilliseconds = 0) | (operationFlags <> 0) then
		detailCode := 5;
	elsif diagnosticsBuild <> 1 then
		detailCode := 16;
	elsif (currentBootId = 0) | (bootId <> currentBootId) then
		detailCode := 17;
	elsif mapRevision <> LMC_DIAG_MAP_REVISION then
		detailCode := 18;
	elsif requestedMode <> 8 then
		detailCode := 45;
	else
		detailCode := 49;
	end_if;
	(pResponse + 12)^$UDINT := detailCode;

END_FUNCTION

FUNCTION LMCDiagnosticsService::HandleAxisSetOperationModeRetire
	VAR_INPUT
		Reference 	: UINT;
		pRequest 	: ^USINT;
		pResponse 	: ^USINT;
		ResponseCapacity 	: UDINT;
		CallerSessionEpoch 	: UDINT;
		RequestSize 	: UDINT;
	END_VAR
	VAR_OUTPUT
		ResponseSize 	: DINT;
	END_VAR
	VAR
		schemaVersion, requestFlags, keySchema, keyReserved : UINT;
		requestId, diagnosticsBuild, bootId, mapRevision : UDINT;
		originalRequestId, intent0, intent1, intent2, intent3 : UDINT;
		timeoutMilliseconds, operationFlags, recordGeneration : UDINT;
		currentBootId, detailCode : UDINT;
		requestedMode : SINT;
		axisReference : UINT;
		reservedByte : USINT;
	END_VAR

	ResponseSize := -1;
	if (pResponse = NIL) | (ResponseCapacity < 16) then
		RETURN;
	end_if;
	_memset(dest:=pResponse, usByte:=0, cntr:=16);
	pResponse^$UINT := LMC_DIAG_SCHEMA_VERSION;
	(pResponse + 4)^$UINT := 1;
	(pResponse + 6)^$INT := LMC_DIAG_ADMIN_ERROR_ID;
	detailCode := 5;
	requestId := 0;
	if (pRequest <> NIL) & (RequestSize >= 8) then
		requestId := (pRequest + 4)^$UDINT;
	end_if;
	(pResponse + 8)^$UDINT := requestId;
	ResponseSize := 16;

	if (pRequest = NIL) | (RequestSize <> 60) then
		(pResponse + 12)^$UDINT := detailCode;
		RETURN;
	end_if;
	schemaVersion := pRequest^$UINT;
	requestFlags := (pRequest + 2)^$UINT;
	keySchema := (pRequest + 8)^$UINT;
	keyReserved := (pRequest + 10)^$UINT;
	diagnosticsBuild := (pRequest + 12)^$UDINT;
	bootId := (pRequest + 16)^$UDINT;
	mapRevision := (pRequest + 20)^$UDINT;
	originalRequestId := (pRequest + 24)^$UDINT;
	intent0 := (pRequest + 28)^$UDINT;
	intent1 := (pRequest + 32)^$UDINT;
	intent2 := (pRequest + 36)^$UDINT;
	intent3 := (pRequest + 40)^$UDINT;
	axisReference := (pRequest + 44)^$UINT;
	requestedMode := (pRequest + 46)^$SINT;
	reservedByte := (pRequest + 47)^$USINT;
	timeoutMilliseconds := (pRequest + 48)^$UDINT;
	operationFlags := (pRequest + 52)^$UDINT;
	recordGeneration := (pRequest + 56)^$UDINT;
	currentBootId := GetDiagnosticsBootId();

	if (schemaVersion <> 1) | (keySchema <> 1) then
		detailCode := 1;
	elsif requestFlags <> 0 then
		detailCode := 2;
	elsif requestId = 0 then
		detailCode := 3;
	elsif (Reference < 1) | (Reference > 4) |
	      (axisReference <> Reference) then
		detailCode := 4;
	elsif (keyReserved <> 0) | (reservedByte <> 0) |
	      (originalRequestId = 0) |
	      ((intent0 = 0) & (intent1 = 0) &
	       (intent2 = 0) & (intent3 = 0)) |
	      (timeoutMilliseconds = 0) | (operationFlags <> 0) |
	      (recordGeneration = 0) then
		detailCode := 5;
	elsif diagnosticsBuild <> 1 then
		detailCode := 16;
	elsif (currentBootId = 0) | (bootId <> currentBootId) then
		detailCode := 17;
	elsif mapRevision <> LMC_DIAG_MAP_REVISION then
		detailCode := 18;
	elsif requestedMode <> 8 then
		detailCode := 45;
	else
		detailCode := 49;
	end_if;
	(pResponse + 12)^$UDINT := detailCode;

END_FUNCTION

FUNCTION LMCDiagnosticsService::ProcessAxisSetOperationMode

END_FUNCTION
